FUNCTION_BLOCK ILOCK_CONFLICT_TRIP_AX (* Prioritizes the first active input and trips on conflict. Requires RESET (Adapter Version). *)
  (* Standard: 61499-2; Description: Copyright (c) 2023 HR Agrartechnik GmbH This program and the accompanying materials are made available under the terms of the Eclipse Public License 2.0 which is available at https://www.eclipse.org/legal/epl-2.0/ SPDX-License-Identifier: EPL-2.0 *)
  (* Version 1.0, 2026-04-19, Franz Höpfinger, HR Agrartechnik GmbH, initial API and implementation and/or initial documentation *)
  PACKAGE logiBUS::signalprocessing::interlock;
  IMPORT eclipse4diac::core::TypeHash;
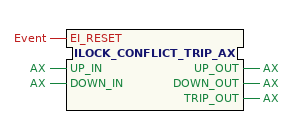
  EVENT_INPUT
    EI_RESET;
  END_EVENT
  SOCKETS
    UP_IN : adapter::types::unidirectional::AX; (* Input for forward/up direction *)
    DOWN_IN : adapter::types::unidirectional::AX; (* Input for backward/down direction *)
  END_SOCKETS
  PLUGS
    UP_OUT : adapter::types::unidirectional::AX; (* Output for forward/up direction *)
    DOWN_OUT : adapter::types::unidirectional::AX; (* Output for backward/down direction *)
    TRIP_OUT : adapter::types::unidirectional::AX; (* Trip State Output *)
  END_PLUGS
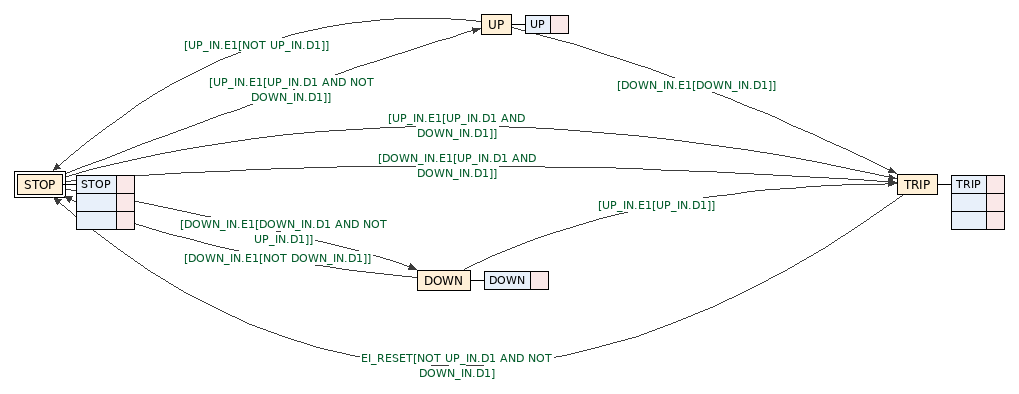
  EC_STATES
    STOP : STOP;
    UP : UP;
    DOWN : DOWN;
    TRIP : TRIP;
  END_STATES
  EC_TRANSITIONS
    STOP TO UP := [UP_IN.E1[UP_IN.D1 AND NOT DOWN_IN.D1]];
    STOP TO DOWN := [DOWN_IN.E1[DOWN_IN.D1 AND NOT UP_IN.D1]];
    STOP TO TRIP := [UP_IN.E1[UP_IN.D1 AND DOWN_IN.D1]];
    STOP TO TRIP := [DOWN_IN.E1[UP_IN.D1 AND DOWN_IN.D1]];
    UP TO STOP := [UP_IN.E1[NOT UP_IN.D1]];
    UP TO TRIP := [DOWN_IN.E1[DOWN_IN.D1]];
    DOWN TO STOP := [DOWN_IN.E1[NOT DOWN_IN.D1]];
    DOWN TO TRIP := [UP_IN.E1[UP_IN.D1]];
    TRIP TO STOP := EI_RESET[NOT UP_IN.D1 AND NOT DOWN_IN.D1];
  END_TRANSITIONS
  ALGORITHM UP IN ST:
UP_OUT.D1 := BOOL#TRUE;
DOWN_OUT.D1 := BOOL#FALSE;
TRIP_OUT.D1 := BOOL#FALSE;
  END_ALGORITHM
  ALGORITHM DOWN IN ST:
UP_OUT.D1 := BOOL#FALSE;
DOWN_OUT.D1 := BOOL#TRUE;
TRIP_OUT.D1 := BOOL#FALSE;
  END_ALGORITHM
  ALGORITHM STOP IN ST:
UP_OUT.D1 := BOOL#FALSE;
DOWN_OUT.D1 := BOOL#FALSE;
TRIP_OUT.D1 := BOOL#FALSE;
  END_ALGORITHM
  ALGORITHM TRIP IN ST:
UP_OUT.D1 := BOOL#FALSE;
DOWN_OUT.D1 := BOOL#FALSE;
TRIP_OUT.D1 := BOOL#TRUE;
  END_ALGORITHM
END_FUNCTION_BLOCK
